Fanuc KAREL source: kt00574.KL

PROGRAM KT00574
%STACKSIZE=65535
%PRIORITY=65535
%NOLOCKGROUP
VAR
R1 : REAL
V2 : VECTOR
OUT : VECTOR
BEGIN
R1=2.0
V2.Y=2.0
-- UNRESOLVED_PC line 10 opcodes [21 49 90 4A] marker_code=36
END KT00574
